{attribute 'qualified_only'}
{attribute 'strict'}
TYPE E_RobotMode :
(
	STOP := 0,
	ESTOP,
	POSITION,
	VELOCITY,
	TORQUE
);
END_TYPE

(* stored: Version 1.1.0.1, ProductVersion 3.1.4024.9
   DUT E_RobotMode: Id {db494ded-5119-4829-9668-a22c486cb433} *)
